(* CoDeSys 2.3.9.472 project: Can 8203 Layer 2.pro *)
(* Libraries: WagoCANLayer2_02.lib 23.6.14 12:08:28, Standard.lib 20.5.14 07:13:26, Iecsfc.lib 16.5.13 13:00:50, SYSLIBCALLBACK.LIB 16.5.13 13:00:50 *)

(* PLC configuration (modules and I/O channels)
Modbus variables [PFC200MODBUS] node 1, in %IB0 out %QB0 {PlcStopBehaviour = 1; FiledbusErrorBehaviour = 1; TcpOperation = 1; TcpPort = 502; TcpTimeout = 600; UdpOperation = 1; UdpPort = 502; RtuOperation = 0; NodeId = 1; ResponseTimeout = 5000; Interface = 0; Baud = 115200; StopBits = 1; Parity = 1; FlowCtrl = 0; PhysInterface = 0}
CAN Layer2 Device [PFC200CANLAYER2] node 2, in %IB6000 out %QB6000 {PFC200CanLayer2NONE = 0}
Modbus-Master [MB_MASTER] node 3, in %IB0 out %QB0
*)

(* Task configuration *)
TASK MainTask (PRIORITY := 6, INTERVAL := T#10ms);
	PLC_PRG();
END_TASK

(* POU PLC_PRG, ST *)
PROGRAM PLC_PRG
VAR
	xOpenPort			: BOOL;
	fbOpenPort		: CAN_OPEN;
	xPortIsOpen		: BOOL;
	fbCanSend			: CAN_TX_29BIT_FRAME :=(
		CAN_ID			:= 16#00000123,
		RTR_FRAME		:= FALSE,
		DATALENGTH	:= 8 );
	fbCanRecv			: CAN_RX_29BIT_FRAME :=(
		CAN_ID			:= 16#00000456,
		CAN_BUFFER	:= FALSE );
	xWrite				: BOOL;
	xRead					: BOOL;
	wState				: WORD;
	aSendData			: ARRAY [1..8] OF BYTE;
	aRecvData			: ARRAY [1..8] OF BYTE;
	bRecvLen			: BYTE;
	tSend					: TON :=(
		PT					:= t#100ms );
END_VAR
fbOpenPort(BAUDRATE:= 125000, ENABLE:= xOpenPort);

fbCanSend(
	DATA:= aSendData,
	ENABLE:= xPortIsOpen,
	WRITE_FRAME:= xWrite );

fbCanRecv(
	ENABLE:= xPortIsOpen,
	READ_FRAME:= xRead );

CASE wState OF
0: (* open CAN port *)
	xOpenPort := TRUE;
	IF fbOpenPort.CONFIRM AND fbOpenPort.ERROR = CAN_PORT_OK THEN
		xOpenPort := FALSE;
		xPortIsOpen := TRUE;
		wState := 10;
	END_IF
10: (* send cyclic messages and check if message was received *)
	tSend(IN := TRUE AND NOT xWrite);
	IF tSend.Q THEN (* sending message *)
		tSend(IN := FALSE);
		xWrite := TRUE;
	ELSIF NOT xRead THEN (* message received *)
		IF fbCanRecv.ERROR = CAN_RECEIVE_OK THEN
			aRecvData := fbCanRecv.DATA;
			bRecvLen := fbCanRecv.DATALENGTH;
			xRead := TRUE;
		ELSE
			xRead := TRUE;
		END_IF
	END_IF
END_CASE
END_PROGRAM

(* POU Configuration/MODBUS_CONFIGURATION, ST *)
PROGRAM MODBUS_CONFIGURATION        
VAR                                
END_VAR                            
(*                                 
   <?xml version="1.0" encoding="UTF-16" standalone="yes"?>
<network xml_structure_version="1" xml_feature_version="1">
	<generator_settings minRTUTaskCycleTimeMs="5" minEthaskCycleTimeMs="5" ethSlaveMultiplier="0.1" rtuInterfaceMultiplier="0.1" taskGeneration="true"/>
</network>
                              
*)                                 
;                                  
END_PROGRAM
